{attribute 'qualified_only'}
{attribute 'to_string'}
TYPE E_CONFIG_STATE :
(
	NO_INIT,
  IDLE,
  INIT_START  := 10,
  INIT_CHECK,
  INIT_DONE,

  READ_START  := 20,
  READ_CHECK,
  READ_DONE,

  WRITE_START := 30,
  WRITE_DONE,

  BUSY        :=  100,
  ERROR       :=  900,
  DONE        := 1000
)UINT;
END_TYPE

(* stored: Version 1.1.0.1, ProductVersion 3.1.4024.13
   DUT E_CONFIG_STATE: Id {5355f1aa-b307-4180-9807-2883f19abacf} *)
